# EPICS IOC start-up script: examples/test/PSI/ep1816-3008.iocsh
#- mXsXXX naming
require ecmccfg,  "NAMING=mXsXXX"

#- add slaves
${SCRIPTEXEC} ${ecmccfg_DIR}addSlave.cmd, "HW_DESC=EP1816-3008, SLAVE_ID=5"

#- apply hardware configuration
${SCRIPTEXEC} ${ecmccfg_DIR}applyConfig.cmd
